PROGRAM MAIN
VAR
	StateMachine: StateMachine;
	fbServer : FB_TCPServer;
	
	SrvNetId : STRING := '';
	ServerPort : UDINT := 9999;
	ServerAddress : STRING := '192.168.108.47';
	
	SResponse : STRING;
	SCommand : STRING;
	Received_data : STRING;
	
	Busy : BOOL;
	Error : BOOL;
	ErrId : UDINT;
	
	Toggle_Timer :TON;
	Mem_Bit AT %MX0.0 : BOOL :=FALSE;
END_VAR

StateMachine();

fbServer(
	send_data:= SResponse, 
	NetId:= SrvNetId, 
	Server_Address:= ServerAddress, 
	Server_Port:= ServerPort, 
	Busy=> Busy, 
	Error=> Error, 
	Received_Data=> SCommand, 
	ErrId=> ErrId);

Toggle_Timer(IN:= NOT Toggle_Timer.Q, PT:= T#1000MS);
Mem_Bit := Toggle_Timer.ET > T#500MS;

SResponse := SCommand;

IF SCommand = 'bit_status' THEN
	IF Mem_Bit THEN
		SResponse := 'BIT ON';
	ELSE
		SResponse := 'BIT OFF';
	END_IF
END_IF

END_PROGRAM

(* stored: Version 1.1.0.1, ProductVersion 3.1.4024.12
   POU MAIN: Id {572507de-a44a-4a7e-b7eb-52f2373576ea}, SpecialFunc None *)
